{attribute 'qualified_only'}
{attribute 'strict'}
{attribute 'to_string'}
TYPE E_EM_LogicExample1_Seq_StartingProduction :
(
	Idle	:= c_nSeqIdle,
	Start	:= c_nSeqStart,
	
	ReferenceAxes,
	CamAxis,
	
	Ready := c_nSeqReady,
	Error := c_nSeqError
);
END_TYPE

(* stored: Version 1.1.0.1, ProductVersion 3.1.4024.10
   DUT E_EM_LogicExample1_Seq_StartingProduction: Id {d76c1092-9297-4317-8feb-7dc5f6a481c2} *)
